// TIA Portal V18 export
// export: Created 2025-12-01T12:38:49.2100586Z, ExportSetting None, DisplayName Totally Integrated Automation Portal, DisplayVersion V18 Update 5, DisplayName TIA Portal Openness, DisplayVersion V18 Update 5, DisplayName TIA Portal Teamcenter Gateway, DisplayVersion V18, DisplayName TIA Portal Version Control Interface, DisplayVersion V18, DisplayName STEP 7 Professional, DisplayVersion V18 Update 5, DisplayName STEP 7 Safety, DisplayVersion V18, DisplayName WinCC Professional, DisplayVersion V18 Update 5
DATA_BLOCK "ST10_FB_S7connect_IDB"   // DB900
// stored: AutoNumber false, InstanceOfName ST10_FB_S7connect, InstanceOfType FB
"ST10_FB_S7connect"
   // VAR_INPUT
   //    "CLOCK_0.2_SEC" : Bool;
   // END_VAR
   // VAR
   //    Always_On : Bool;
   //    Status_Get : Array[1..6] of Struct
   //       NDR : Bool;
   //       Error : Bool;
   //       Status : Int;
   //    END_STRUCT;
   //    Status_Put : Array[1..6] of Struct
   //       Done : Bool;
   //       Error : Bool;
   //       Status : Int;
   //    END_STRUCT;
   //    GET_Instance1 { S7_SetPoint := 'True'} : GET;
   //    GET_Instance2 { S7_SetPoint := 'True'} : GET;
   //    PUT_Instance1 { S7_SetPoint := 'True'} : PUT;
   //    PUT_Instance2 { S7_SetPoint := 'True'} : PUT;
   //    PLs { S7_SetPoint := 'True'} : Array[1..6] of Bool;
   //    TON : Array[1..5] of TON_TIME;
   //    NextStation_OffLine : Bool;
   // END_VAR
BEGIN
END_DATA_BLOCK
